Staubli VAL3: moveTo.pgx

program moveTo(trsf x_trMoveTo (dimensions=1), config x_cMoveTo (dimensions=1), num& x_nFlagStep[] (dimensions=1))
  local bool l_bResult
  local num l_nKeyPressed
  local num l_nMotionStatus
  local num l_nState
  local point l_pMoveTo
begin
  l_pMoveTo=here(tPointer,world)
  // Check workingmode (must be in jog/Point)
  workingMode(l_nState)
  if (l_nState>0) and (l_nState!=nMANUAL_HOLD)
    call up:msgBox(lang:sListOfMessage[40+l_nState],36,lang:sMenu[1],l_nKeyPressed)
    x_nFlagStep=-1
  else
    l_pMoveTo.trsf=x_trMoveTo
    l_pMoveTo.config=x_cMoveTo
    taskCreate "motion",20,moveRobot(l_pMoveTo)
    // wait until task is created
    wait(taskStatus("motion")==1)
    do
      l_nMotionStatus=taskStatus("motion")
    until (l_nMotionStatus==-1) or (l_nMotionStatus>1)
    // started task stopped because of run-rime error
    if l_nMotionStatus>1
      taskKill("motion")
      wait(taskStatus("motion")==-1)
    elseIf nMotionError!=0
      call up:msgBox(sErrorMessage,36,lang:sMenu[1],l_nKeyPressed)
      x_nFlagStep=-1
      nMotionError=0
    endIf
  endIf
end
